Omron CX-Programmer project NewProject (CX-Programmer 9.75)

# PLC NewPLC1: CP1E N60

## Global symbols (name address type ; comment)
A_Pulse 0.00 BOOL
Appr_PX 0.04 BOOL  ; 0.04
AutoCycle 4 NUMBER  ; 4
105 CHANNEL  ; AO1
108 CHANNEL  ; AO4
A531.00 BOOL  ; =
D1201 CHANNEL  ; Run Hrs
D1202 CHANNEL  ; Auto Cycle Count
D901 CHANNEL  ; AO4_DA_Val
D902 CHANNEL  ; PS_ValC
D904 CHANNEL  ; PS_DA_Val
D905 CHANNEL  ; MaxPSVal
D908 CHANNEL  ; .
D910 CHANNEL  ; UnlockPS
D911 CHANNEL  ; ApprPrePS
D912 CHANNEL  ; ApprPS
D913 CHANNEL  ; Pressing PS
D915 CHANNEL  ; TRUpPS
D916 CHANNEL  ; EjPS
H0 CHANNEL  ; Run Sec
H1 CHANNEL  ; Run Minute
H2 CHANNEL  ; Run Hr
T025 BOOL  ; Min Press2
W10.05 BOOL  ; Decomp PS
AutoMan_SS 2.03 BOOL  ; 2.03 1=Auto
AutoON_PB1 1.02 BOOL  ; 1.02
AutoON_PB2 1.03 BOOL  ; 1.03
AutoReady 3 NUMBER  ; 3
AutoSTDBY 2 NUMBER  ; 2
B_Pulse 0.01 BOOL
DoorCloseSOL 102.06 BOOL  ; 102.06
DoorOpenSOL 102.05 BOOL  ; 102.05
Door_Close_PB 2.02 BOOL  ; 2.02
Door_Open_PB 2.01 BOOL  ; 2.01
Door_Open_PX 0.09 BOOL  ; 0.09
Drive_RO3 2.07 BOOL  ; 2.07
Ej_A2T_SOL 102.07 BOOL  ; 102.07
Ej_DN_SOL 102.00 BOOL  ; 102.00
Ej_Up_SOL 101.00 BOOL  ; 101.00
EjectDN_PB 2.00 BOOL  ; 2.00
EjectDN_PX 0.10 BOOL  ; 0.10
EjectMID_PX 0.11 BOOL  ; 0.11
EjectUP_PB 1.11 BOOL  ; 1.11
EjectUP_PX 1.00 BOOL  ; 1.0
ExtTrig 109.05 BOOL  ; 102.05
FLocked_PX 0.05 BOOL  ; 0.05
F_LockRel_PX 0.06 BOOL  ; 0.06
LockState 6 NUMBER  ; 6
Lock_PB 1.09 BOOL  ; 1.09
Lock_SOL 101.03 BOOL  ; 101.03
MainUL_SOL 101.02 BOOL  ; 101.02
Main_HP_UL 101.01 BOOL  ; 101.01
Manual 1 NUMBER  ; 1
MotorOFF_PB 1.06 BOOL  ; 1.06
MotorON_PB 1.05 BOOL  ; 1.05
OffState 0 NUMBER  ; 0
OilLow_PX 1.01 BOOL  ; 1.01
PG_SR 2.08 BOOL  ; 2.08
PMD_Fault 2.06 BOOL  ; 2.06
PilotPumpON 102.04 BOOL  ; 102.04
PilotUnloadSOL 102.01 BOOL  ; 102.01
Pilot_CBOK 2.05 BOOL  ; 2.05
Pilot_CV_SOL 100.05 BOOL  ; 100.05
Pilot_DN_SOL 101.04 BOOL  ; 101.04
Pilot_UP_SOL 100.01 BOOL  ; 100.01
Prefill_SOL 100.07 BOOL  ; 100.07
PulsOut1 100.00 BOOL  ; Puls1_OUT
PulsOut1_Dir 100.02 BOOL
RLocked_PX 0.07 BOOL  ; 0.07
R_LockRel_PX 0.08 BOOL  ; 0.08
SK1_Off 2.09 BOOL  ; SK1_FB
SK2_Off 2.10 BOOL  ; 2.10
TR_DN_PB 1.08 BOOL  ; 1.08
TR_DN_PX 0.03 BOOL  ; 0.03
TR_Home_PX 0.02 BOOL  ; 0.02
TR_Pres_SOL 101.05 BOOL  ; 101.05
TR_UP_PB 1.07 BOOL  ; 1.07
TileEject 5 NUMBER  ; 5
TileEject_PB 1.04 BOOL  ; 1.04
Unlock_PB 1.10 BOOL  ; 1.10
Unlock_SOL 100.04 BOOL  ; 100.04
Water_CBOK 2.04 BOOL  ; 2.04

## Program NewProgram1 (cyclic task 0)
Local symbols
AP_PS_bar D104 WORD  ; D104
AP_Pre_PS D116 WORD  ; D116
AP_Pre_RPM D117 WORD  ; D117
AReq_Seq1 W51.00 BOOL  ; W51.0
A_DoorDN W52.09 BOOL  ; W52.09
A_DoorUP W52.08 BOOL  ; W52.08
A_EJ_DN W52.05 BOOL  ; W52.05
A_EJ_UP W52.04 BOOL  ; W52.04
A_Ej_B2t W52.14 BOOL  ; W52.14
A_Lock W52.06 BOOL  ; W52.06
A_MotorON W52.01 BOOL  ; W52.01
A_PilotCV W52.11 BOOL  ; W52.11
A_PilotDN W52.12 BOOL  ; W52.12
A_PrefilSOL W52.10 BOOL  ; W52.10
A_Seq1 W50.00 BOOL  ; W50.0
A_Seq10 W50.09 BOOL  ; W50.09
A_Seq11 W50.10 BOOL  ; W50.10
A_Seq12 W50.11 BOOL  ; W50.11
A_Seq13 W50.12 BOOL  ; W50.12
A_Seq14 W50.13 BOOL  ; W50.13
A_Seq15 W50.14 BOOL  ; W50.14
A_Seq16 W50.15 BOOL  ; W50.15
A_Seq2 W50.01 BOOL  ; W50.01
A_Seq3 W50.02 BOOL  ; W50.02
A_Seq4 W50.03 BOOL  ; W50.03
A_Seq5 W50.04 BOOL  ; W50.04
A_Seq6 W50.05 BOOL  ; W50.05
A_Seq7 W50.06 BOOL  ; W50.06
A_Seq8 W50.07 BOOL  ; W50.07
A_Seq9 W50.08 BOOL  ; W50.08
A_SeqWD W50 WORD  ; W50
A_TR_DN W52.02 BOOL  ; W52.02
A_TR_UP W52.03 BOOL  ; W52.03
A_Unlock W52.07 BOOL  ; W52.07
ApprRPM D103 WORD  ; D103
Appr_PX_ERR W41.05 BOOL  ; W41.05
AutoReqSeq W51 WORD  ; W51
Auto_PBSimul D571 WORD  ; D571
Auto_PBTim D572 WORD  ; D572
BR_PX_SIMUL W41.01 BOOL  ; W41.01
DOOR_PX_SIMUL W41.02 BOOL  ; W41.02
DeComp1Tim D111 WORD  ; D111
Decomp1TMR T015 BOOL  ; T15
Decomp2TMR T017 BOOL  ; T17
Decomp2Tim D113 WORD  ; D113
DieModeON W49.00 BOOL  ; W49.00
Die_Bypass W49.01 BOOL  ; W49.01
DoorOpen_UNLOCK W41.06 BOOL  ; W41.06
EJ_MID_PX_FAIL W41.03 BOOL  ; W41.03
EjUP_Seq1 W53.00 BOOL  ; W53.00
EjUP_Seq2 W53.01 BOOL  ; W53.01
EjUP_Seq3 W53.02 BOOL  ; W53.02
EjUP_Seq4 W53.03 BOOL  ; W53.03
EjUpSPD D109 WORD  ; D109
EjectWtTMR T014 BOOL  ; T14
Eject_Wt D108 WORD  ; d108
FastApprTMR T022 BOOL  ; T22
HMI_AutoCycle W56.10 BOOL  ; W56.10
HMI_AutoRDY W56.09 BOOL  ; W56.09
HMI_Door_Down W57.08 BOOL  ; W57.08
HMI_Door_Down_PX W58.12 BOOL  ; W58.12
HMI_Door_Mid W58.11 BOOL  ; W58.11
HMI_Door_Op_PX W58.10 BOOL  ; W58.10
HMI_Door_UP W57.07 BOOL  ; W57.07
HMI_DriveFault W56.06 BOOL  ; W56.06
HMI_EJ_DN_PX W58.08 BOOL  ; W58.08
HMI_EJ_Down W57.06 BOOL  ; W57.06
HMI_EJ_MID_PX W58.09 BOOL  ; W58.09
HMI_EJ_UP W57.05 BOOL  ; W57.05
HMI_EJ_UP_PX W58.07 BOOL  ; W58.07
HMI_EStop W56.03 BOOL  ; W56.03
HMI_FUL_PX W58.01 BOOL  ; W58.01
HMI_Float W56.01 BOOL  ; W56.01
HMI_Flock_PX W58.00 BOOL  ; W58.00
HMI_LockState W56.04 BOOL
HMI_Lock_Sol W57.09 BOOL  ; W57.09
HMI_M_DoorClose_PB W60.00 BOOL  ; W60.0
HMI_M_DoorOpen_PB W58.15 BOOL
HMI_M_EJ_DN_PB W60.02 BOOL  ; W60.02
HMI_M_EJ_UP_PB W60.01 BOOL  ; W60.01
HMI_M_Lock_PB W58.14 BOOL  ; W58.14
HMI_M_TR_DN W60.04 BOOL  ; W60.04
HMI_M_TR_UP_PB W60.03 BOOL  ; W60.03
HMI_M_Unlock_PB W58.13 BOOL  ; W58.13
HMI_Main_M_ON W56.11 BOOL  ; W56.11
HMI_Main_UL W57.01 BOOL  ; W57.01
HMI_PG_Clear W56.08 BOOL  ; W56.08
HMI_Phase W56.02 BOOL  ; W56.02
HMI_Pilot_M_ON W56.12 BOOL  ; w56.12
HMI_Pilot_OLR W56.00 BOOL  ; W56.0
HMI_Pilot_UL W57.00 BOOL  ; W57.00
HMI_Pre_SOL W57.12 BOOL  ; W57.12
HMI_Pressing_Sol W57.11 BOOL  ; W57.11
HMI_RUL_PX W58.03 BOOL  ; W58.03
HMI_Rlock_PX W58.02 BOOL  ; W58.02
HMI_STO W56.07 BOOL  ; W56.07
HMI_TR_AP_PX W58.05 BOOL  ; W58.05
HMI_TR_CV W57.02 BOOL  ; W57.02
HMI_TR_DN_PX W58.06 BOOL  ; W58.06
HMI_TR_Down W57.04 BOOL  ; W57.04
HMI_TR_Home W58.04 BOOL  ; W58.04
HMI_TR_UP W57.03 BOOL  ; W57.03
HMI_Unlock_Sol W57.10 BOOL  ; W57.10
HMI_WaterOLR W56.05 BOOL  ; W56.05
HandIn W53.04 BOOL  ; w53.04
LockRPM D107 WORD  ; D107
Lock_PX_SIMUL W41.04 BOOL  ; W41.04
MAXSV D560 CHANNEL  ; D560
MAXSV_bar D610 WORD  ; D610
MAXSV_w D561 CHANNEL  ; D561
MINSV D550 CHANNEL  ; D550
MINSV_w D551 CHANNEL  ; D551
M_DoorDN W40.09 BOOL
M_DoorUP W40.08 BOOL
M_EJ_DN W40.05 BOOL
M_EJ_UP W40.04 BOOL
M_Lock W40.06 BOOL
M_MotorON W40.01 BOOL
M_TR_DN W40.02 BOOL
M_TR_UP W40.03 BOOL
M_Unlock W40.07 BOOL
ManualRPM D570 WORD  ; D570
MinApprTMR T012 BOOL  ; T12
MinApprTim D105 WORD  ; D105
MinPress1Tim D115 WORD  ; D115
MinPressTMR T018 BOOL  ; T18
MotorSPD D510 WORD  ; D510
PS W10.00 BOOL  ; Pressure
PS2 T016 BOOL  ; PS2
PS2_Add D112 WORD  ; D112
PS_2 W10.02 BOOL  ; W10.02
PS_Appr W10.01 BOOL
PS_Appr_Pre W10.04 BOOL  ; W10.04
PS_ERR W10.12 BOOL  ; W10.12
PS_Pre W10.03 BOOL  ; W10.03
PS_Pre_Bar D613 WORD  ; D613
PS_Pre_SV D612 WORD  ; D612
PV_bar D602 CHANNEL  ; D602
PV_in D601 CHANNEL  ; D601
PV_remind D603 CHANNEL  ; D603
Pr_MAX_D1 D1100 WORD  ; D1100
Pr_MAX_D2 D1101 WORD  ; D1101
PressRPM D110 WORD  ; D110
PressRPMPre D114 WORD  ; D114
Ps_Bar D900 CHANNEL  ; D900
SV2_add D607 WORD  ; D607
SV2_bar D609 WORD  ; D609
SV2_remind D608 WORD  ; d608
SV_bar D604 CHANNEL  ; D604
SV_in D600 CHANNEL  ; D600
SV_remind D605 CHANNEL  ; D605
Simult_OK W55.02 BOOL  ; Simult OK
SpinUpTMR T010 BOOL  ; T10
SpinUpTim D102 WORD
SpinupTMR T011 BOOL  ; T11
TE_DoorDN W52.09 BOOL  ; W60.00
TE_DoorUP W52.08 BOOL  ; W60.01
TE_EJ_DN W52.05 BOOL  ; W60.02
TE_EJ_UP W52.04 BOOL  ; W60.03
TRUpSPD D106 WORD  ; D106
TR_DN_PX_Sense W55.04 BOOL  ; W55.04
TR_DN_Sensed W55.04 BOOL  ; W55.04
TR_PX_SIMUL W41.00 BOOL  ; W41.00
TileEJSeq W54 WORD  ; W54
TileEJ_DN W54.00 BOOL  ; W54.0
Tile_Ej_Mode W55.03 BOOL  ; W55.03
UnlockRPM D101 WORD  ; D101
UnlockSlowRPM D118 WORD  ; D118
m_MainMotor_ON W12.00 BOOL  ; W12.0
min_appr D105 WORD  ; min_appr
st_AutoCycle W16.04 BOOL
st_AutoReady W16.03 BOOL
st_AutoSTDBY W16.02 BOOL
st_LockState W16.06 BOOL  ; W16.06
st_Manual W16.01 BOOL
st_Off W16.00 BOOL
st_TileEject W16.05 BOOL
state D700 CHANNEL  ; D700
sto_rec_tim D100 WORD  ; sto_rec_tim

### Section States

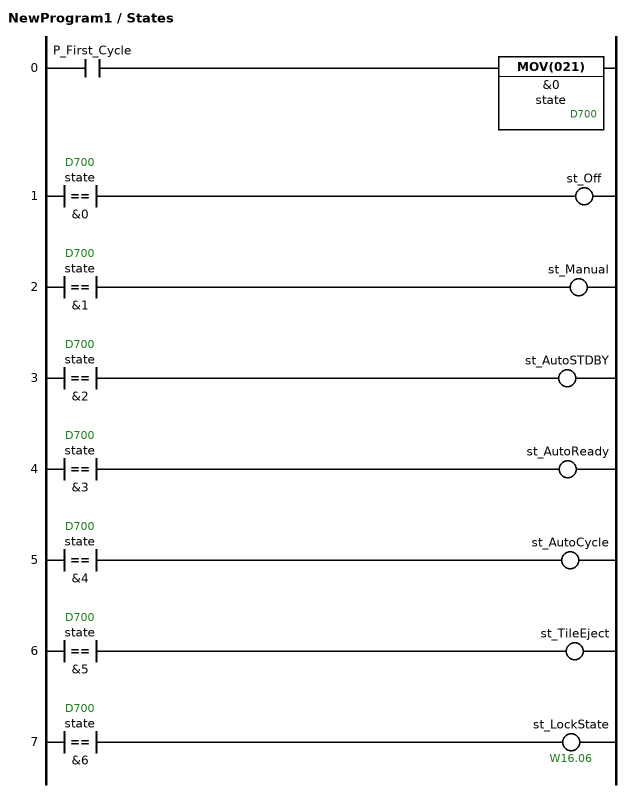
; rung 0
LD P_First_Cycle
MOV(021) &0 state  ; D700
; rung 1
LD=(300) state &0  ; D700
OUT st_Off
; rung 2
LD=(300) state &1  ; D700
OUT st_Manual
; rung 3
LD=(300) state &2  ; D700
OUT st_AutoSTDBY
; rung 4
LD=(300) state &3  ; D700
OUT st_AutoReady
; rung 5
LD=(300) state &4  ; D700
OUT st_AutoCycle
; rung 6
LD=(300) state &5  ; D700
OUT st_TileEject
; rung 7
LD=(300) state &6  ; D700
OUT st_LockState  ; W16.06

### Section IO

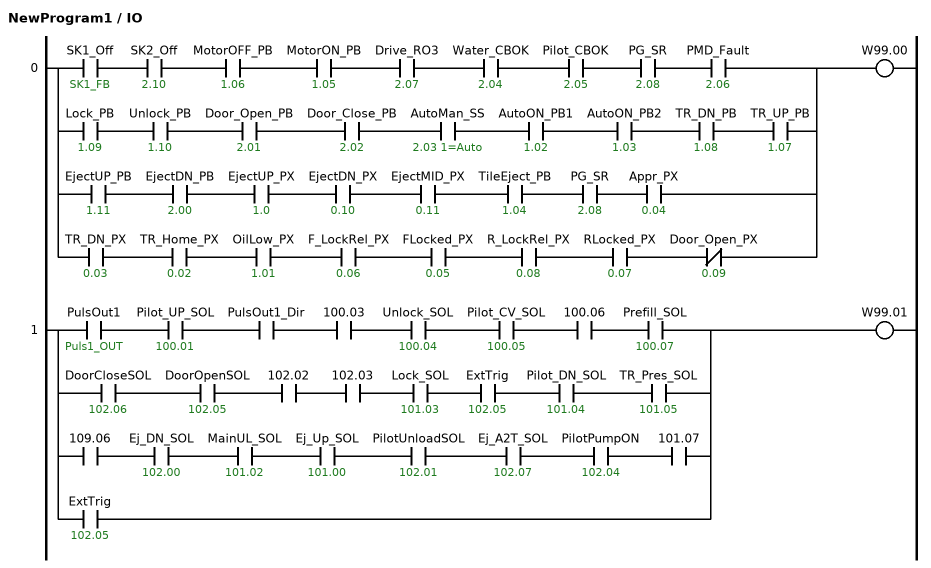
; rung 0
LD SK1_Off  ; SK1_FB
AND SK2_Off  ; 2.10
AND MotorOFF_PB  ; 1.06
AND MotorON_PB  ; 1.05
AND Drive_RO3  ; 2.07
AND Water_CBOK  ; 2.04
AND Pilot_CBOK  ; 2.05
AND PG_SR  ; 2.08
AND PMD_Fault  ; 2.06
LD Lock_PB  ; 1.09
AND Unlock_PB  ; 1.10
AND Door_Open_PB  ; 2.01
AND Door_Close_PB  ; 2.02
AND AutoMan_SS  ; 2.03 1=Auto
AND AutoON_PB1  ; 1.02
AND AutoON_PB2  ; 1.03
AND TR_DN_PB  ; 1.08
AND TR_UP_PB  ; 1.07
ORLD
LD EjectUP_PB  ; 1.11
AND EjectDN_PB  ; 2.00
AND EjectUP_PX  ; 1.0
AND EjectDN_PX  ; 0.10
AND EjectMID_PX  ; 0.11
AND TileEject_PB  ; 1.04
AND PG_SR  ; 2.08
AND Appr_PX  ; 0.04
ORLD
LD TR_DN_PX  ; 0.03
AND TR_Home_PX  ; 0.02
AND OilLow_PX  ; 1.01
AND F_LockRel_PX  ; 0.06
AND FLocked_PX  ; 0.05
AND R_LockRel_PX  ; 0.08
AND RLocked_PX  ; 0.07
ANDNOT Door_Open_PX  ; 0.09
ORLD
OUT W99.00
; rung 1
LD PulsOut1  ; Puls1_OUT
AND Pilot_UP_SOL  ; 100.01
AND PulsOut1_Dir
AND 100.03
AND Unlock_SOL  ; 100.04
AND Pilot_CV_SOL  ; 100.05
AND 100.06
AND Prefill_SOL  ; 100.07
LD DoorCloseSOL  ; 102.06
AND DoorOpenSOL  ; 102.05
AND 102.02
AND 102.03
AND Lock_SOL  ; 101.03
AND ExtTrig  ; 102.05
AND Pilot_DN_SOL  ; 101.04
AND TR_Pres_SOL  ; 101.05
ORLD
LD 109.06
AND Ej_DN_SOL  ; 102.00
AND MainUL_SOL  ; 101.02
AND Ej_Up_SOL  ; 101.00
AND PilotUnloadSOL  ; 102.01
AND Ej_A2T_SOL  ; 102.07
AND PilotPumpON  ; 102.04
AND 101.07
ORLD
OR ExtTrig  ; 102.05
OUT W99.01

### Section PressureControl

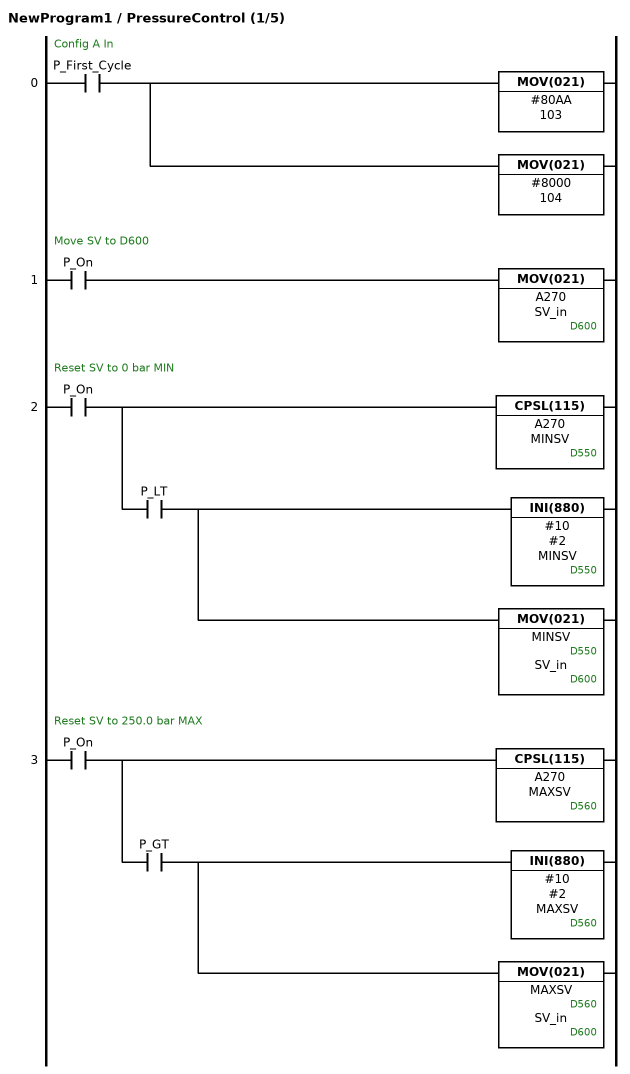
; rung 0: Config A In
LD P_First_Cycle
MOV(021) #80AA 103
MOV(021) #8000 104
; rung 1: Move SV to D600
LD P_On
MOV(021) A270 SV_in  ; D600
; rung 2: Reset SV to 0 bar MIN
LD P_On
CPSL(115) A270 MINSV  ; D550
AND P_LT
INI(880) #10 #2 MINSV  ; D550
MOV(021) MINSV SV_in  ; D550, D600
; rung 3: Reset SV to 250.0 bar MAX
LD P_On
CPSL(115) A270 MAXSV  ; D560
AND P_GT
INI(880) #10 #2 MAXSV  ; D560
MOV(021) MAXSV SV_in  ; D560, D600

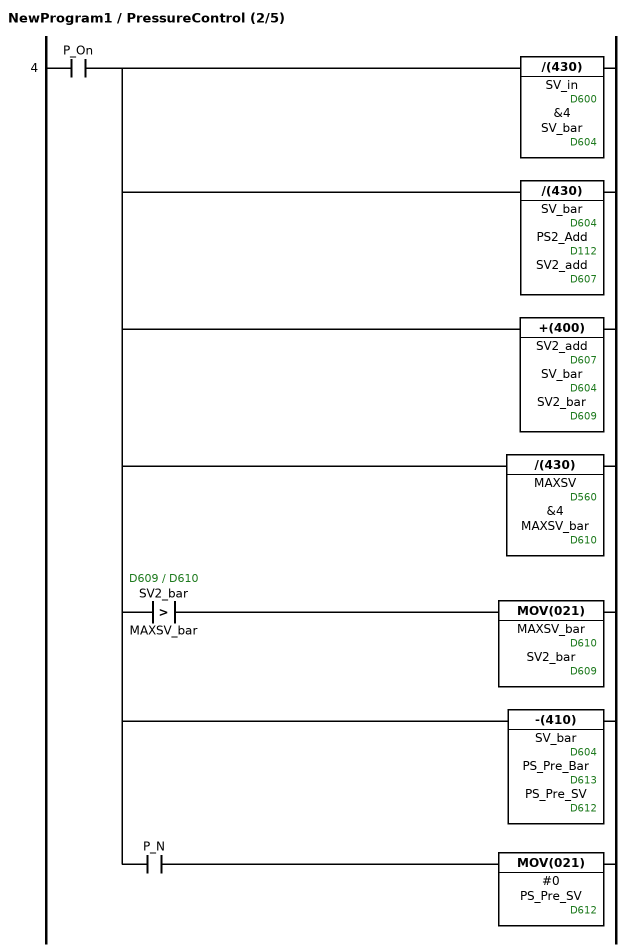
; rung 4
LD P_On
OUT TR0
/(430) SV_in &4 SV_bar  ; D600, D604
/(430) SV_bar PS2_Add SV2_add  ; D604, D112, D607
+(400) SV2_add SV_bar SV2_bar  ; D607, D604, D609
/(430) MAXSV &4 MAXSV_bar  ; D560, D610
AND>(320) SV2_bar MAXSV_bar  ; D609, D610
MOV(021) MAXSV_bar SV2_bar  ; D610, D609
LD TR0
-(410) SV_bar PS_Pre_Bar PS_Pre_SV  ; D604, D613, D612
AND P_N
MOV(021) #0 PS_Pre_SV  ; D612

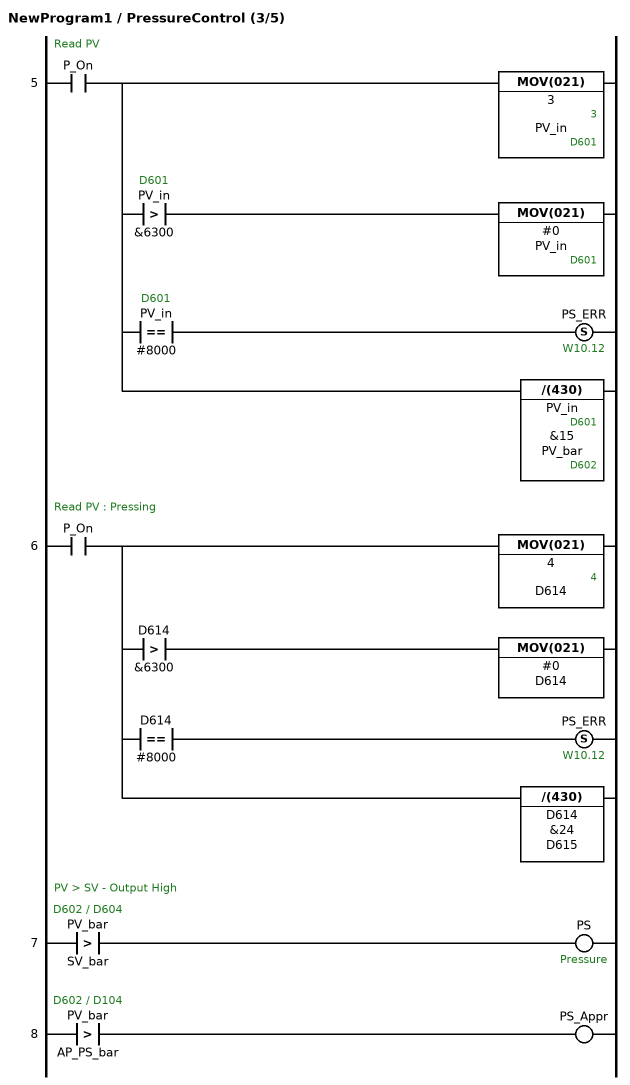
; rung 5: Read PV
LD P_On
OUT TR0
MOV(021) 3 PV_in  ; 3, D601
AND>(320) PV_in &6300  ; D601
MOV(021) #0 PV_in  ; D601
LD TR0
AND=(300) PV_in #8000  ; D601
SET PS_ERR  ; W10.12
LD TR0
/(430) PV_in &15 PV_bar  ; D601, D602
; rung 6: Read PV : Pressing
LD P_On
OUT TR0
MOV(021) 4 D614  ; 4
AND>(320) D614 &6300
MOV(021) #0 D614
LD TR0
AND=(300) D614 #8000
SET PS_ERR  ; W10.12
LD TR0
/(430) D614 &24 D615
; rung 7: PV > SV - Output High
LD>(320) PV_bar SV_bar  ; D602, D604
OUT PS  ; Pressure
; rung 8
LD>(320) PV_bar AP_PS_bar  ; D602, D104
OUT PS_Appr

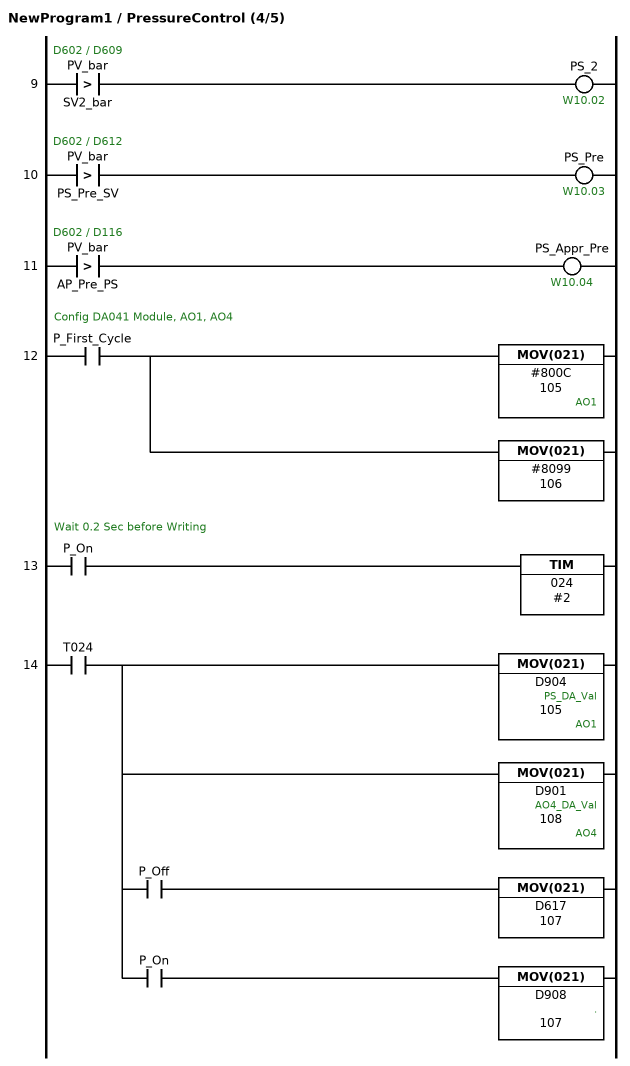
; rung 9
LD>(320) PV_bar SV2_bar  ; D602, D609
OUT PS_2  ; W10.02
; rung 10
LD>(320) PV_bar PS_Pre_SV  ; D602, D612
OUT PS_Pre  ; W10.03
; rung 11
LD>(320) PV_bar AP_Pre_PS  ; D602, D116
OUT PS_Appr_Pre  ; W10.04
; rung 12: Config DA041 Module, AO1, AO4
LD P_First_Cycle
MOV(021) #800C 105  ; AO1
MOV(021) #8099 106
; rung 13: Wait 0.2 Sec before Writing
LD P_On
TIM 024 #2
; rung 14
LD T024
OUT TR0
MOV(021) D904 105  ; PS_DA_Val, AO1
MOV(021) D901 108  ; AO4_DA_Val, AO4
AND P_Off
MOV(021) D617 107
LD TR0
AND P_On
MOV(021) D908 107  ; .

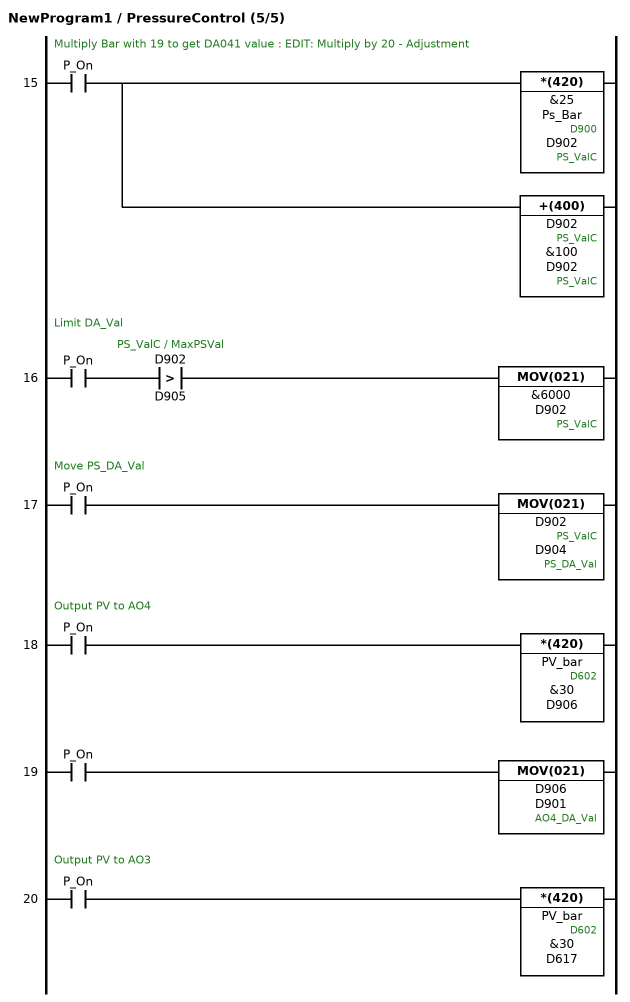
; rung 15: Multiply Bar with 19 to get DA041 value : EDIT: Multiply by 20 - Adjustment
LD P_On
*(420) &25 Ps_Bar D902  ; D900, PS_ValC
+(400) D902 &100 D902  ; PS_ValC
; rung 16: Limit DA_Val
LD P_On
AND>(320) D902 D905  ; PS_ValC, MaxPSVal
MOV(021) &6000 D902  ; PS_ValC
; rung 17: Move PS_DA_Val
LD P_On
MOV(021) D902 D904  ; PS_ValC, PS_DA_Val
; rung 18: Output PV to AO4
LD P_On
*(420) PV_bar &30 D906  ; D602
; rung 19
LD P_On
MOV(021) D906 D901  ; AO4_DA_Val
; rung 20: Output PV to AO3
LD P_On
*(420) PV_bar &30 D617  ; D602

### Section OFFState

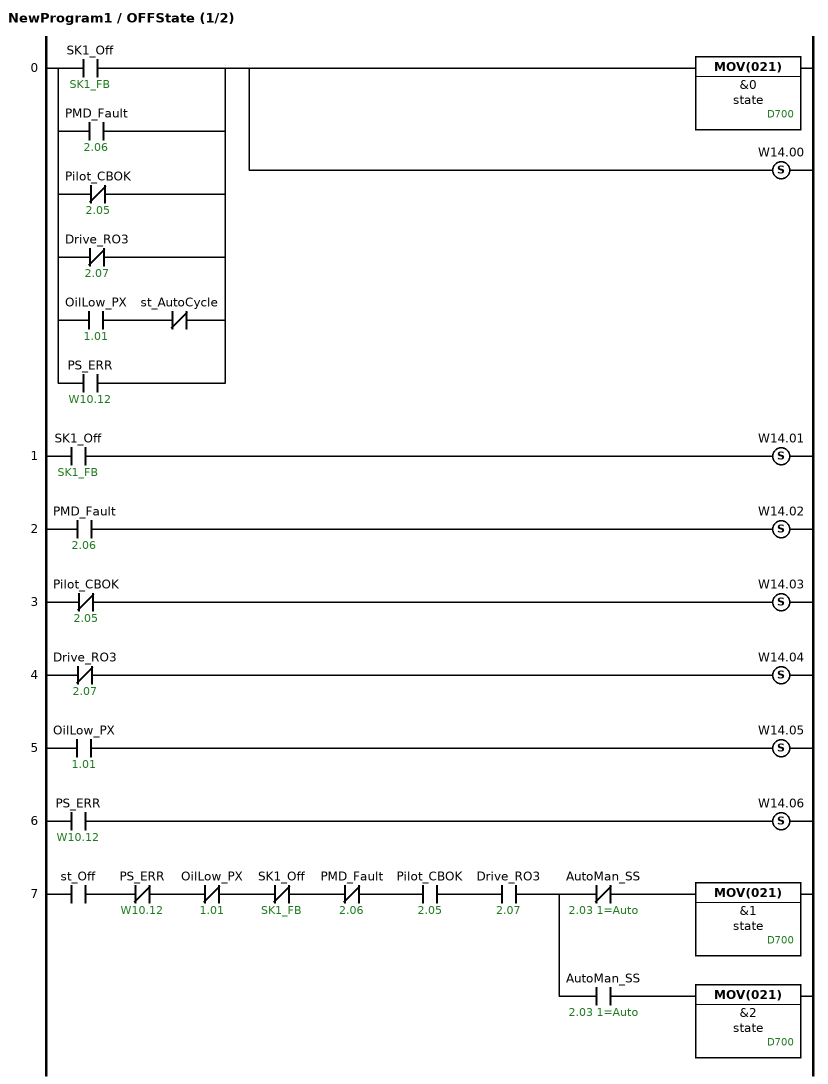
; rung 0
LD SK1_Off  ; SK1_FB
OR PMD_Fault  ; 2.06
ORNOT Pilot_CBOK  ; 2.05
ORNOT Drive_RO3  ; 2.07
LD OilLow_PX  ; 1.01
ANDNOT st_AutoCycle
ORLD
OR PS_ERR  ; W10.12
MOV(021) &0 state  ; D700
SET W14.00
; rung 1
LD SK1_Off  ; SK1_FB
SET W14.01
; rung 2
LD PMD_Fault  ; 2.06
SET W14.02
; rung 3
LDNOT Pilot_CBOK  ; 2.05
SET W14.03
; rung 4
LDNOT Drive_RO3  ; 2.07
SET W14.04
; rung 5
LD OilLow_PX  ; 1.01
SET W14.05
; rung 6
LD PS_ERR  ; W10.12
SET W14.06
; rung 7
LD st_Off
ANDNOT PS_ERR  ; W10.12
ANDNOT OilLow_PX  ; 1.01
ANDNOT SK1_Off  ; SK1_FB
ANDNOT PMD_Fault  ; 2.06
AND Pilot_CBOK  ; 2.05
AND Drive_RO3  ; 2.07
OUT TR0
ANDNOT AutoMan_SS  ; 2.03 1=Auto
MOV(021) &1 state  ; D700
LD TR0
AND AutoMan_SS  ; 2.03 1=Auto
MOV(021) &2 state  ; D700

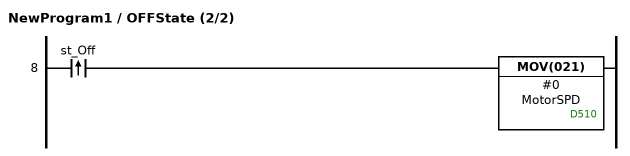
; rung 8
@LD st_Off
MOV(021) #0 MotorSPD  ; D510

### Section LockState

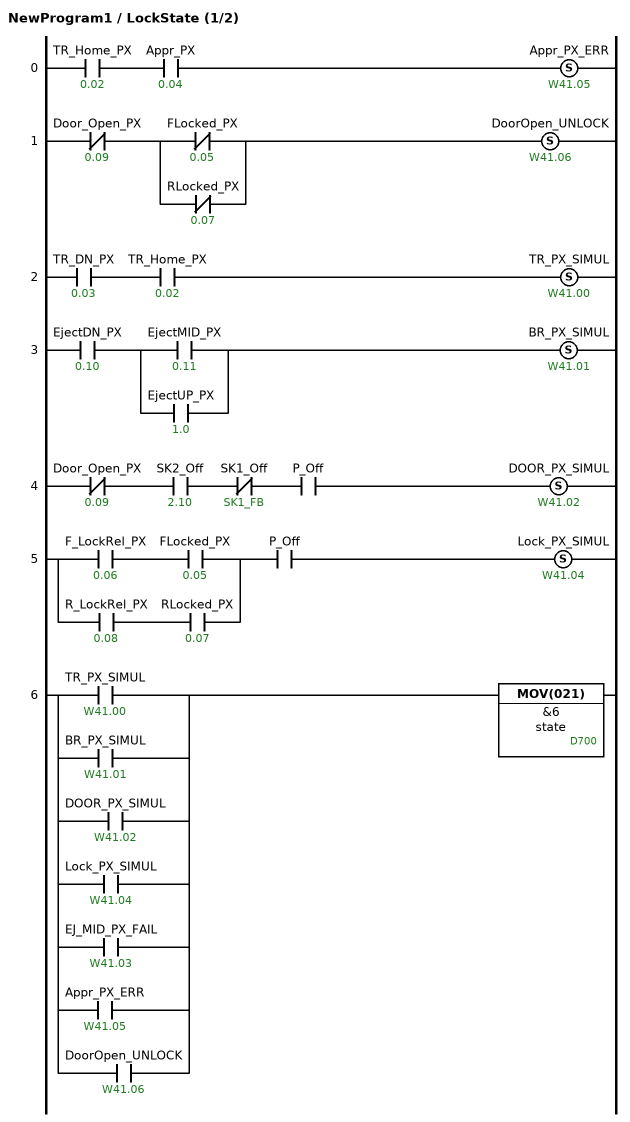
; rung 0
LD TR_Home_PX  ; 0.02
AND Appr_PX  ; 0.04
SET Appr_PX_ERR  ; W41.05
; rung 1
LDNOT Door_Open_PX  ; 0.09
LDNOT FLocked_PX  ; 0.05
ORNOT RLocked_PX  ; 0.07
ANDLD
SET DoorOpen_UNLOCK  ; W41.06
; rung 2
LD TR_DN_PX  ; 0.03
AND TR_Home_PX  ; 0.02
SET TR_PX_SIMUL  ; W41.00
; rung 3
LD EjectDN_PX  ; 0.10
LD EjectMID_PX  ; 0.11
OR EjectUP_PX  ; 1.0
ANDLD
SET BR_PX_SIMUL  ; W41.01
; rung 4
LDNOT Door_Open_PX  ; 0.09
AND SK2_Off  ; 2.10
ANDNOT SK1_Off  ; SK1_FB
AND P_Off
SET DOOR_PX_SIMUL  ; W41.02
; rung 5
LD F_LockRel_PX  ; 0.06
AND FLocked_PX  ; 0.05
LD R_LockRel_PX  ; 0.08
AND RLocked_PX  ; 0.07
ORLD
AND P_Off
SET Lock_PX_SIMUL  ; W41.04
; rung 6
LD TR_PX_SIMUL  ; W41.00
OR BR_PX_SIMUL  ; W41.01
OR DOOR_PX_SIMUL  ; W41.02
OR Lock_PX_SIMUL  ; W41.04
OR EJ_MID_PX_FAIL  ; W41.03
OR Appr_PX_ERR  ; W41.05
OR DoorOpen_UNLOCK  ; W41.06
MOV(021) &6 state  ; D700

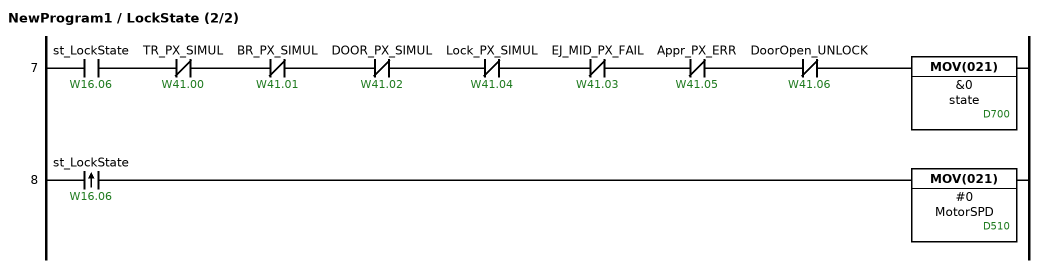
; rung 7
LD st_LockState  ; W16.06
ANDNOT TR_PX_SIMUL  ; W41.00
ANDNOT BR_PX_SIMUL  ; W41.01
ANDNOT DOOR_PX_SIMUL  ; W41.02
ANDNOT Lock_PX_SIMUL  ; W41.04
ANDNOT EJ_MID_PX_FAIL  ; W41.03
ANDNOT Appr_PX_ERR  ; W41.05
ANDNOT DoorOpen_UNLOCK  ; W41.06
MOV(021) &0 state  ; D700
; rung 8
@LD st_LockState  ; W16.06
MOV(021) #0 MotorSPD  ; D510

### Section Manual

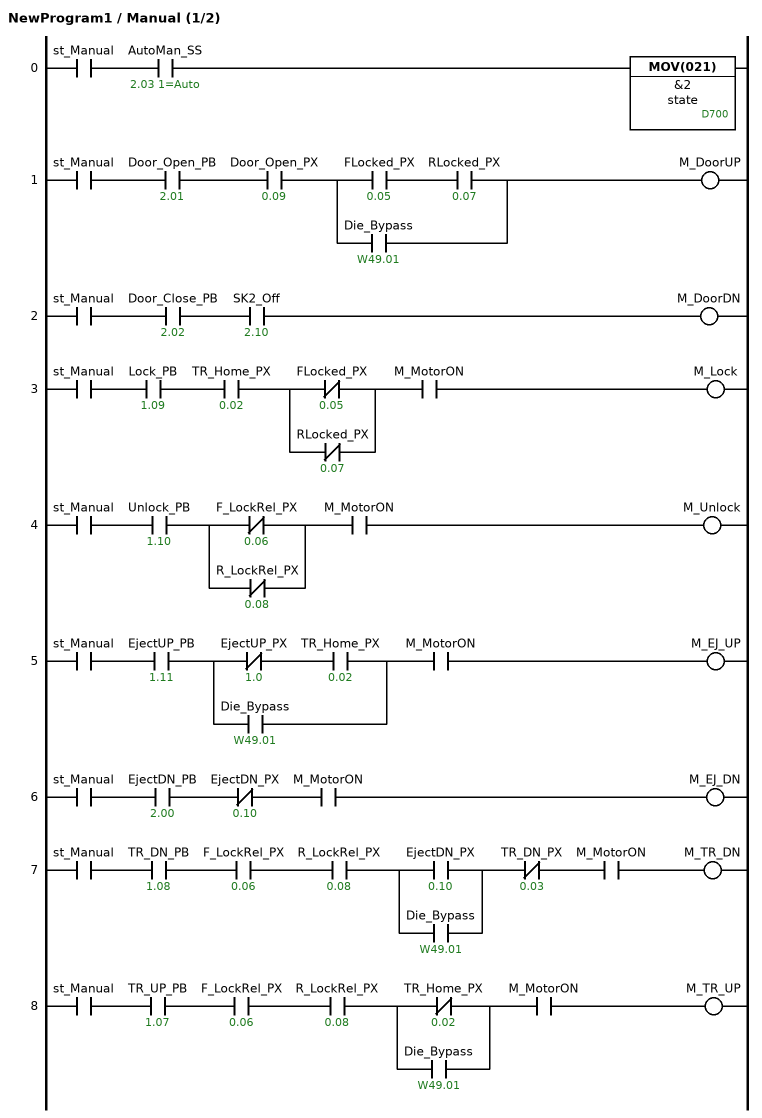
; rung 0
LD st_Manual
AND AutoMan_SS  ; 2.03 1=Auto
MOV(021) &2 state  ; D700
; rung 1
LD st_Manual
AND Door_Open_PB  ; 2.01
AND Door_Open_PX  ; 0.09
LD FLocked_PX  ; 0.05
AND RLocked_PX  ; 0.07
OR Die_Bypass  ; W49.01
ANDLD
OUT M_DoorUP
; rung 2
LD st_Manual
AND Door_Close_PB  ; 2.02
AND SK2_Off  ; 2.10
OUT M_DoorDN
; rung 3
LD st_Manual
AND Lock_PB  ; 1.09
AND TR_Home_PX  ; 0.02
LDNOT FLocked_PX  ; 0.05
ORNOT RLocked_PX  ; 0.07
ANDLD
AND M_MotorON
OUT M_Lock
; rung 4
LD st_Manual
AND Unlock_PB  ; 1.10
LDNOT F_LockRel_PX  ; 0.06
ORNOT R_LockRel_PX  ; 0.08
ANDLD
AND M_MotorON
OUT M_Unlock
; rung 5
LD st_Manual
AND EjectUP_PB  ; 1.11
LDNOT EjectUP_PX  ; 1.0
AND TR_Home_PX  ; 0.02
OR Die_Bypass  ; W49.01
ANDLD
AND M_MotorON
OUT M_EJ_UP
; rung 6
LD st_Manual
AND EjectDN_PB  ; 2.00
ANDNOT EjectDN_PX  ; 0.10
AND M_MotorON
OUT M_EJ_DN
; rung 7
LD st_Manual
AND TR_DN_PB  ; 1.08
AND F_LockRel_PX  ; 0.06
AND R_LockRel_PX  ; 0.08
LD EjectDN_PX  ; 0.10
OR Die_Bypass  ; W49.01
ANDLD
ANDNOT TR_DN_PX  ; 0.03
AND M_MotorON
OUT M_TR_DN
; rung 8
LD st_Manual
AND TR_UP_PB  ; 1.07
AND F_LockRel_PX  ; 0.06
AND R_LockRel_PX  ; 0.08
LDNOT TR_Home_PX  ; 0.02
OR Die_Bypass  ; W49.01
ANDLD
AND M_MotorON
OUT M_TR_UP

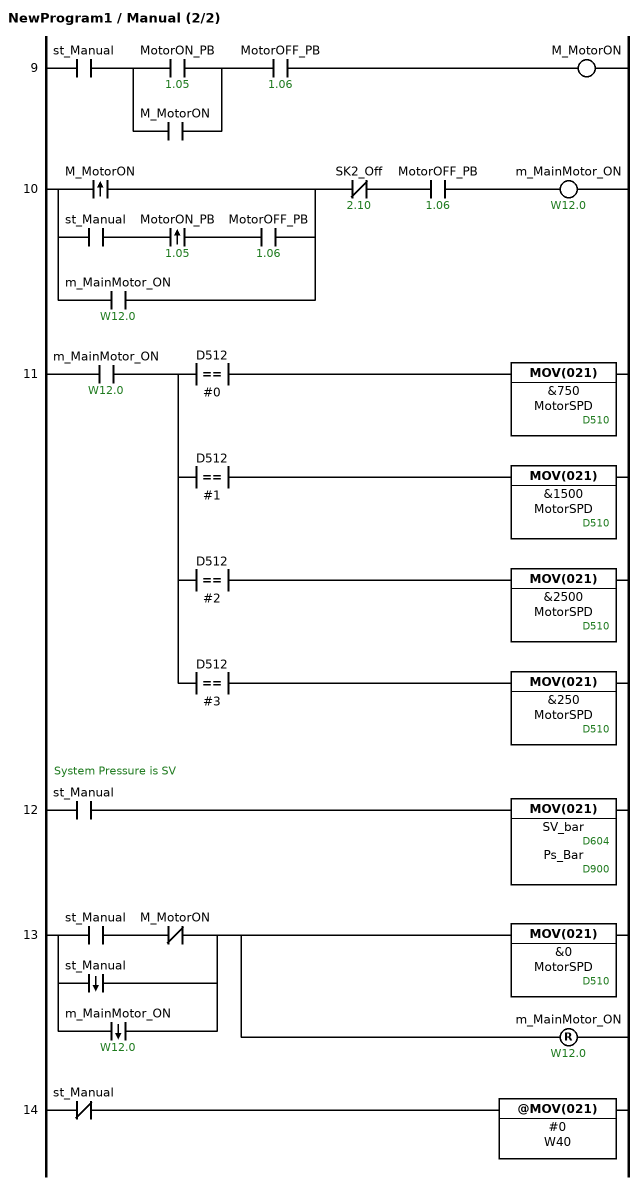
; rung 9
LD st_Manual
LD MotorON_PB  ; 1.05
OR M_MotorON
ANDLD
AND MotorOFF_PB  ; 1.06
OUT M_MotorON
; rung 10
@LD M_MotorON
LD st_Manual
@AND MotorON_PB  ; 1.05
AND MotorOFF_PB  ; 1.06
ORLD
OR m_MainMotor_ON  ; W12.0
ANDNOT SK2_Off  ; 2.10
AND MotorOFF_PB  ; 1.06
OUT m_MainMotor_ON  ; W12.0
; rung 11
LD m_MainMotor_ON  ; W12.0
OUT TR0
AND=(300) D512 #0
MOV(021) &750 MotorSPD  ; D510
LD TR0
AND=(300) D512 #1
MOV(021) &1500 MotorSPD  ; D510
LD TR0
AND=(300) D512 #2
MOV(021) &2500 MotorSPD  ; D510
LD TR0
AND=(300) D512 #3
MOV(021) &250 MotorSPD  ; D510
; rung 12: System Pressure is SV
LD st_Manual
MOV(021) SV_bar Ps_Bar  ; D604, D900
; rung 13
LD st_Manual
ANDNOT M_MotorON
%OR st_Manual
%OR m_MainMotor_ON  ; W12.0
MOV(021) &0 MotorSPD  ; D510
RSET m_MainMotor_ON  ; W12.0
; rung 14
LDNOT st_Manual
@MOV(021) #0 W40

### Section DieMode

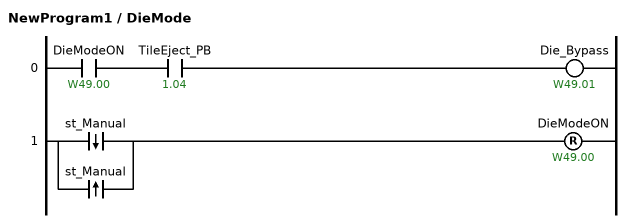
; rung 0
LD DieModeON  ; W49.00
AND TileEject_PB  ; 1.04
OUT Die_Bypass  ; W49.01
; rung 1
%LD st_Manual
@OR st_Manual
RSET DieModeON  ; W49.00

### Section AutoSTDBY

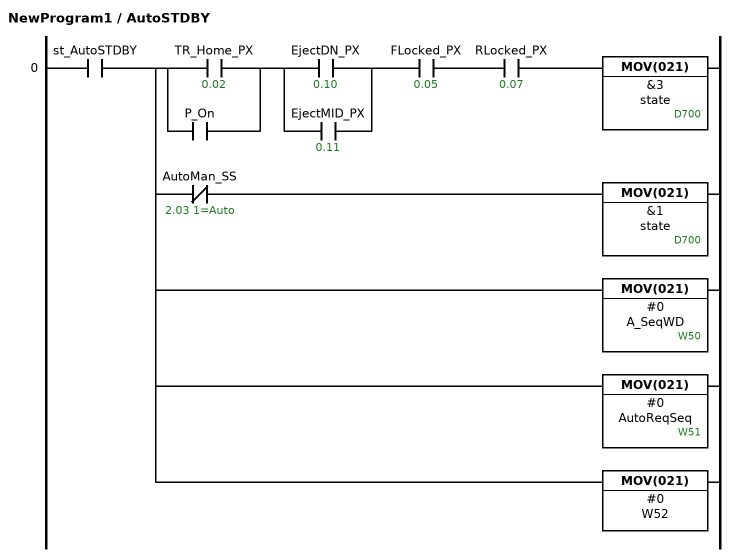
; rung 0
LD st_AutoSTDBY
OUT TR0
LD TR_Home_PX  ; 0.02
OR P_On
ANDLD
LD EjectDN_PX  ; 0.10
OR EjectMID_PX  ; 0.11
ANDLD
AND FLocked_PX  ; 0.05
AND RLocked_PX  ; 0.07
MOV(021) &3 state  ; D700
LD TR0
ANDNOT AutoMan_SS  ; 2.03 1=Auto
MOV(021) &1 state  ; D700
LD TR0
MOV(021) #0 A_SeqWD  ; W50
MOV(021) #0 AutoReqSeq  ; W51
MOV(021) #0 W52

### Section AutoReady

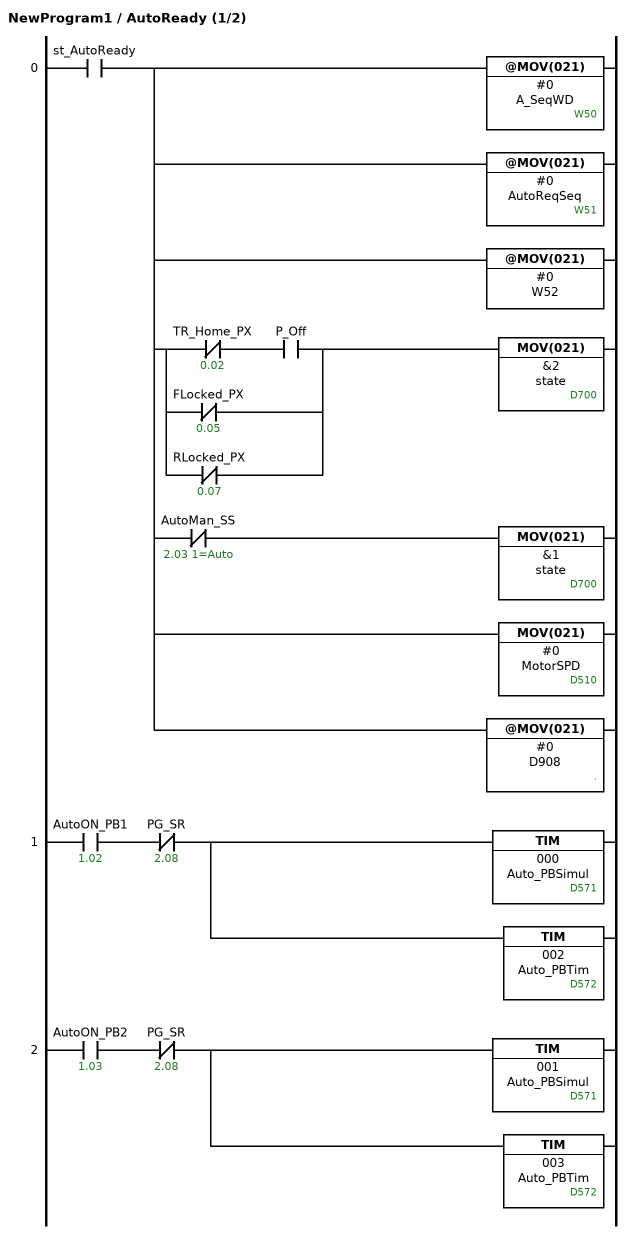
; rung 0
LD st_AutoReady
OUT TR0
@MOV(021) #0 A_SeqWD  ; W50
@MOV(021) #0 AutoReqSeq  ; W51
@MOV(021) #0 W52
LDNOT TR_Home_PX  ; 0.02
AND P_Off
ORNOT FLocked_PX  ; 0.05
ORNOT RLocked_PX  ; 0.07
ANDLD
MOV(021) &2 state  ; D700
LD TR0
ANDNOT AutoMan_SS  ; 2.03 1=Auto
MOV(021) &1 state  ; D700
LD TR0
MOV(021) #0 MotorSPD  ; D510
@MOV(021) #0 D908  ; .
; rung 1
LD AutoON_PB1  ; 1.02
ANDNOT PG_SR  ; 2.08
TIM 000 Auto_PBSimul  ; D571
TIM 002 Auto_PBTim  ; D572
; rung 2
LD AutoON_PB2  ; 1.03
ANDNOT PG_SR  ; 2.08
TIM 001 Auto_PBSimul  ; D571
TIM 003 Auto_PBTim  ; D572

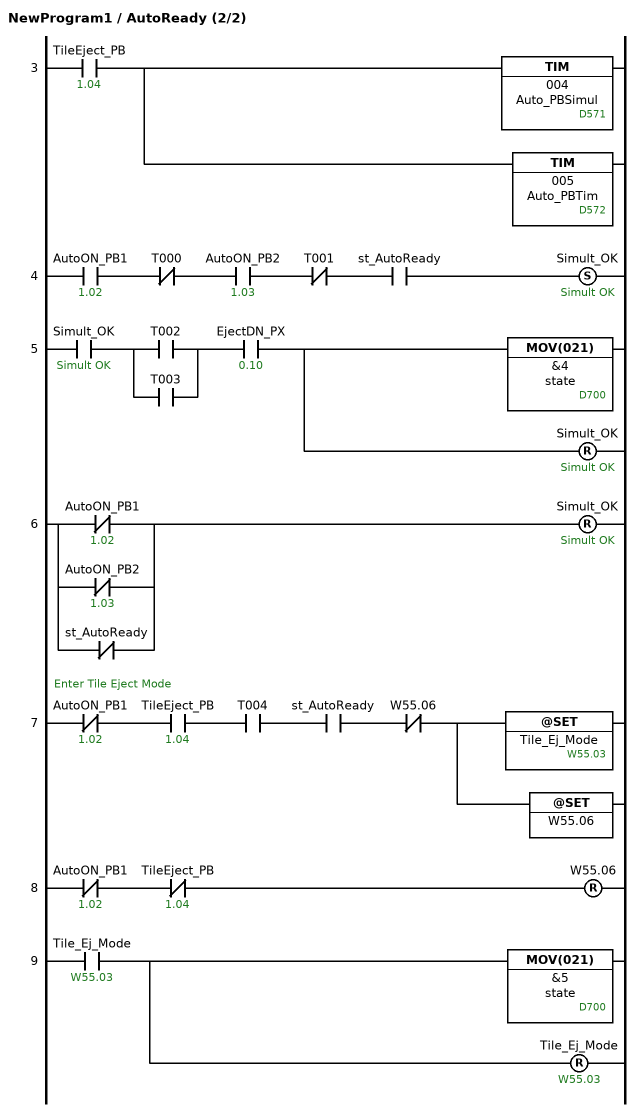
; rung 3
LD TileEject_PB  ; 1.04
TIM 004 Auto_PBSimul  ; D571
TIM 005 Auto_PBTim  ; D572
; rung 4
LD AutoON_PB1  ; 1.02
ANDNOT T000
AND AutoON_PB2  ; 1.03
ANDNOT T001
AND st_AutoReady
SET Simult_OK  ; Simult OK
; rung 5
LD Simult_OK  ; Simult OK
LD T002
OR T003
ANDLD
AND EjectDN_PX  ; 0.10
MOV(021) &4 state  ; D700
RSET Simult_OK  ; Simult OK
; rung 6
LDNOT AutoON_PB1  ; 1.02
ORNOT AutoON_PB2  ; 1.03
ORNOT st_AutoReady
RSET Simult_OK  ; Simult OK
; rung 7: Enter Tile Eject Mode
LDNOT AutoON_PB1  ; 1.02
AND TileEject_PB  ; 1.04
AND T004
AND st_AutoReady
ANDNOT W55.06
@SET Tile_Ej_Mode  ; W55.03
@SET W55.06
; rung 8
LDNOT AutoON_PB1  ; 1.02
ANDNOT TileEject_PB  ; 1.04
RSET W55.06
; rung 9
LD Tile_Ej_Mode  ; W55.03
MOV(021) &5 state  ; D700
RSET Tile_Ej_Mode  ; W55.03

### Section AutoCycle

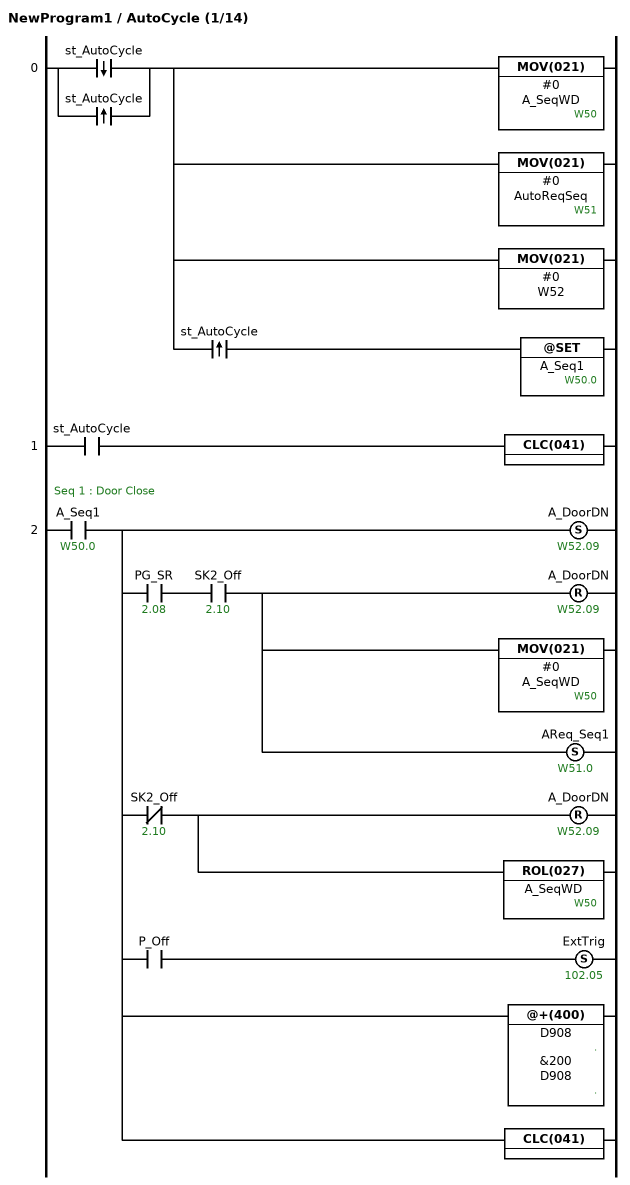
; rung 0
%LD st_AutoCycle
@OR st_AutoCycle
MOV(021) #0 A_SeqWD  ; W50
MOV(021) #0 AutoReqSeq  ; W51
MOV(021) #0 W52
@AND st_AutoCycle
@SET A_Seq1  ; W50.0
; rung 1
LD st_AutoCycle
CLC(041)
; rung 2: Seq 1 : Door Close
LD A_Seq1  ; W50.0
OUT TR0
SET A_DoorDN  ; W52.09
AND PG_SR  ; 2.08
AND SK2_Off  ; 2.10
RSET A_DoorDN  ; W52.09
MOV(021) #0 A_SeqWD  ; W50
SET AReq_Seq1  ; W51.0
LD TR0
ANDNOT SK2_Off  ; 2.10
RSET A_DoorDN  ; W52.09
ROL(027) A_SeqWD  ; W50
LD TR0
AND P_Off
SET ExtTrig  ; 102.05
LD TR0
@+(400) D908 &200 D908  ; .
CLC(041)

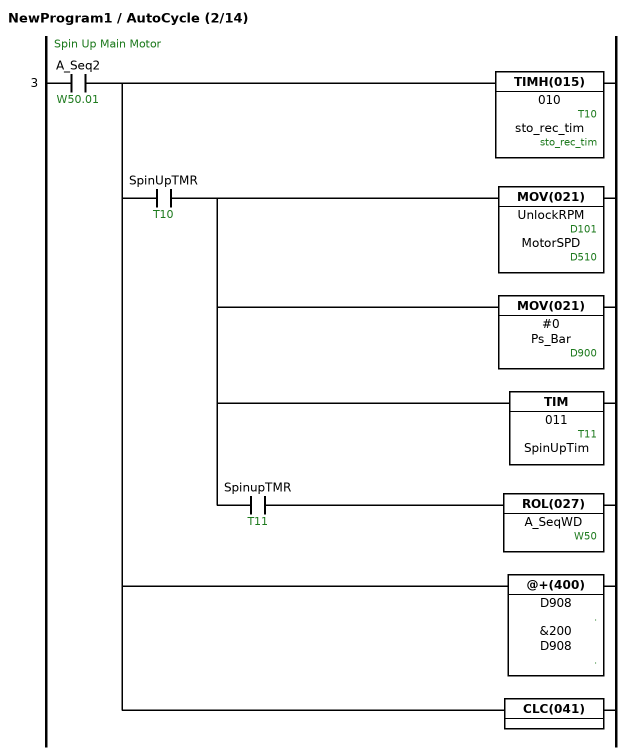
; rung 3: Spin Up Main Motor
LD A_Seq2  ; W50.01
OUT TR0
TIMH(015) 010 sto_rec_tim  ; sto_rec_tim, T10
AND SpinUpTMR  ; T10
MOV(021) UnlockRPM MotorSPD  ; D101, D510
MOV(021) #0 Ps_Bar  ; D900
TIM 011 SpinUpTim  ; T11
AND SpinupTMR  ; T11
ROL(027) A_SeqWD  ; W50
LD TR0
@+(400) D908 &200 D908  ; .
CLC(041)

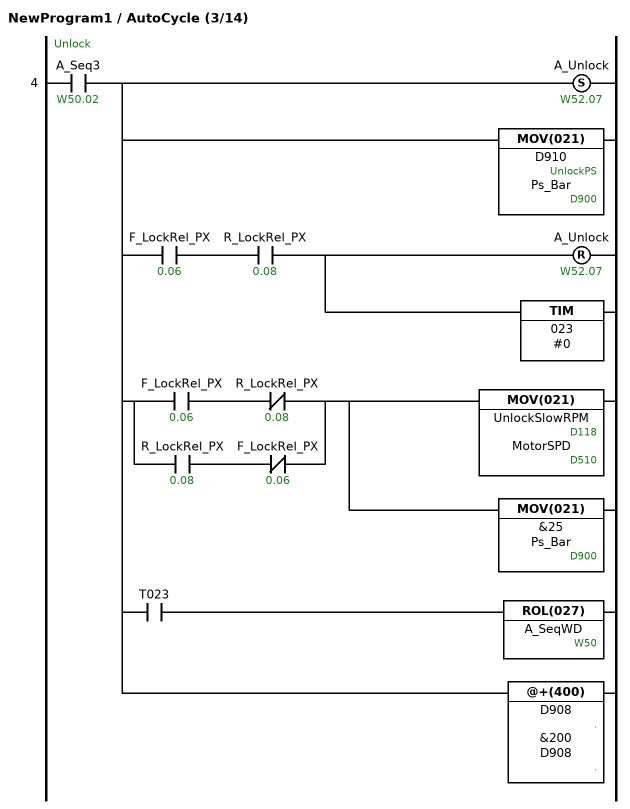
; rung 4: Unlock
LD A_Seq3  ; W50.02
OUT TR0
SET A_Unlock  ; W52.07
MOV(021) D910 Ps_Bar  ; UnlockPS, D900
AND F_LockRel_PX  ; 0.06
AND R_LockRel_PX  ; 0.08
RSET A_Unlock  ; W52.07
TIM 023 #0
LD TR0
LD F_LockRel_PX  ; 0.06
ANDNOT R_LockRel_PX  ; 0.08
LD R_LockRel_PX  ; 0.08
ANDNOT F_LockRel_PX  ; 0.06
ORLD
ANDLD
MOV(021) UnlockSlowRPM MotorSPD  ; D118, D510
MOV(021) &25 Ps_Bar  ; D900
LD TR0
AND T023
ROL(027) A_SeqWD  ; W50
LD TR0
@+(400) D908 &200 D908  ; .

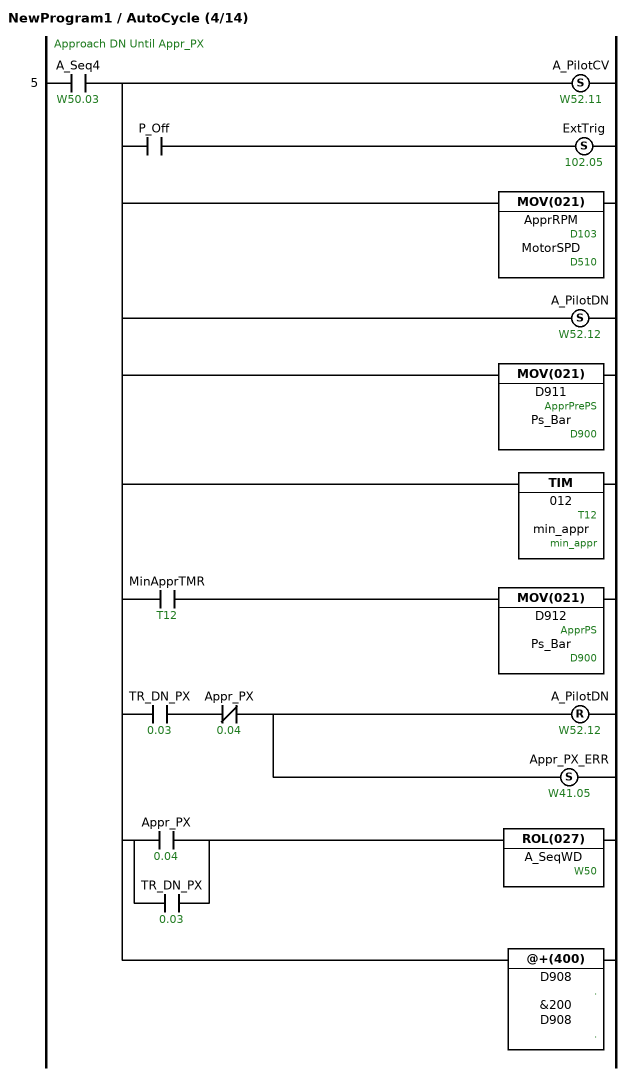
; rung 5: Approach DN Until Appr_PX
LD A_Seq4  ; W50.03
OUT TR0
SET A_PilotCV  ; W52.11
AND P_Off
SET ExtTrig  ; 102.05
LD TR0
MOV(021) ApprRPM MotorSPD  ; D103, D510
SET A_PilotDN  ; W52.12
MOV(021) D911 Ps_Bar  ; ApprPrePS, D900
TIM 012 min_appr  ; min_appr, T12
AND MinApprTMR  ; T12
MOV(021) D912 Ps_Bar  ; ApprPS, D900
LD TR0
AND TR_DN_PX  ; 0.03
ANDNOT Appr_PX  ; 0.04
RSET A_PilotDN  ; W52.12
SET Appr_PX_ERR  ; W41.05
LD TR0
LD Appr_PX  ; 0.04
OR TR_DN_PX  ; 0.03
ANDLD
ROL(027) A_SeqWD  ; W50
LD TR0
@+(400) D908 &200 D908  ; .

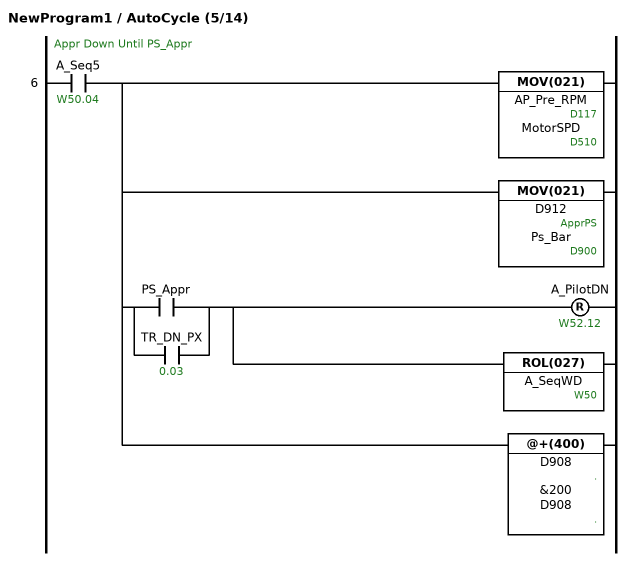
; rung 6: Appr Down Until PS_Appr
LD A_Seq5  ; W50.04
OUT TR0
MOV(021) AP_Pre_RPM MotorSPD  ; D117, D510
MOV(021) D912 Ps_Bar  ; ApprPS, D900
LD PS_Appr
OR TR_DN_PX  ; 0.03
ANDLD
RSET A_PilotDN  ; W52.12
ROL(027) A_SeqWD  ; W50
LD TR0
@+(400) D908 &200 D908  ; .

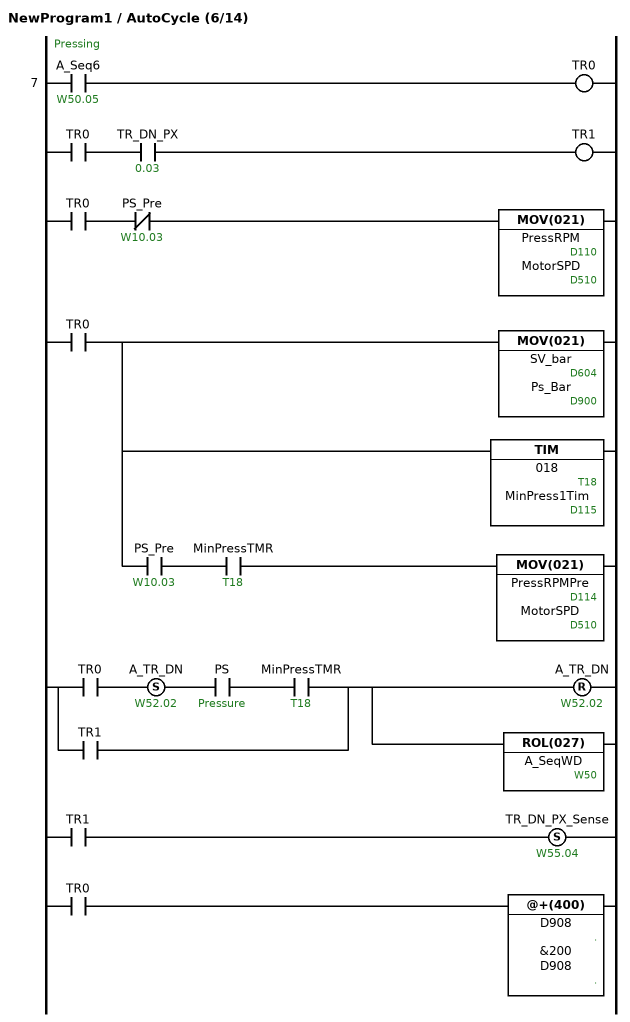
; rung 7: Pressing
LD A_Seq6  ; W50.05
OUT TR0
ANDNOT PS_Pre  ; W10.03
MOV(021) PressRPM MotorSPD  ; D110, D510
LD TR0
MOV(021) SV_bar Ps_Bar  ; D604, D900
TIM 018 MinPress1Tim  ; D115, T18
AND PS_Pre  ; W10.03
AND MinPressTMR  ; T18
MOV(021) PressRPMPre MotorSPD  ; D114, D510
LD TR0
SET A_TR_DN  ; W52.02
AND PS  ; Pressure
AND MinPressTMR  ; T18
LD TR0
AND TR_DN_PX  ; 0.03
OUT TR1
ORLD
RSET A_TR_DN  ; W52.02
ROL(027) A_SeqWD  ; W50
LD TR1
SET TR_DN_PX_Sense  ; W55.04
LD TR0
@+(400) D908 &200 D908  ; .

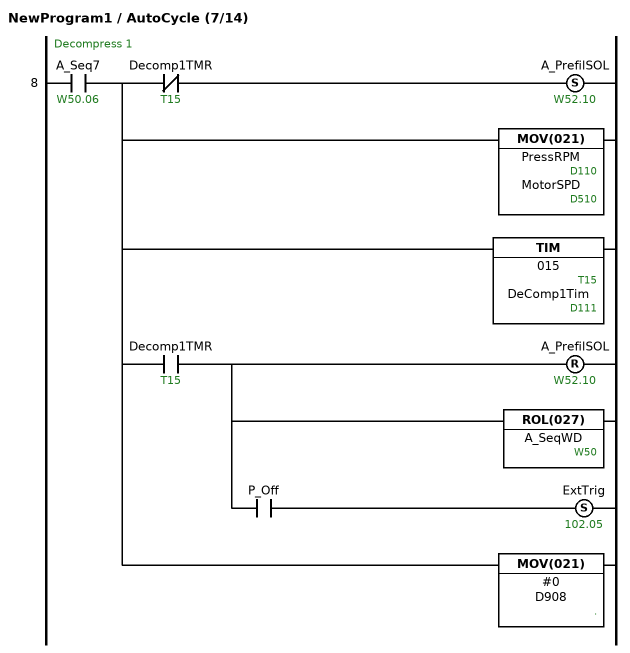
; rung 8: Decompress 1
LD A_Seq7  ; W50.06
OUT TR0
ANDNOT Decomp1TMR  ; T15
SET A_PrefilSOL  ; W52.10
LD TR0
MOV(021) PressRPM MotorSPD  ; D110, D510
TIM 015 DeComp1Tim  ; D111, T15
AND Decomp1TMR  ; T15
RSET A_PrefilSOL  ; W52.10
ROL(027) A_SeqWD  ; W50
AND P_Off
SET ExtTrig  ; 102.05
LD TR0
MOV(021) #0 D908  ; .

